// TIA Portal V15.1 export
// export: Created 2020-06-12T07:35:48.3037109Z, ExportSetting None, DisplayName Totally Integrated Automation Portal, DisplayVersion V15.1, DisplayName TIA Portal Openness, DisplayVersion V15.1, DisplayName STEP 7 Professional, DisplayVersion V15.1, DisplayName STEP 7 Safety, DisplayVersion V15.1, DisplayName WinCC Advanced, DisplayVersion V15.1
FUNCTION "PWR_ctrl" : Void   // FC751, FBD
TITLE = High current line
{ S7_Optimized_Access := 'TRUE' }
// stored: AutoNumber false, SetENOAutomatically False
   VAR_TEMP
      _dummy : Bool;
      _csf : Bool;   // Common system fault
      _trans_release : Bool;
      _mcb_lock : Bool;
      _mcb_start : Bool;
      _mcb_stop : Bool;
      _mcb_stop_cmd : Bool;
      _mcb_save_off : Bool;
      _slag_ok : Bool;
      _sealing_ok : Bool;
      _tp : Time;
      _toff : Bool;
      _spare : Bool;
      tRet : Int;
      tPmax : Real;
      tImax : Real;
      _mcb_released : Bool;
      tCbOn : Bool;
      tCosPhi : Real;
      tSwitchPulse : Bool;
      tCbExtOn : Bool;
      tCbExtOff : Bool;
      tCbIntOff : Bool;
      tCircuitInsulFault : Bool;
      tTrafoCoolFault : Bool;
      tCBisDisabled : Bool;
   END_VAR
BEGIN

REGION Network 1: Common System Fault
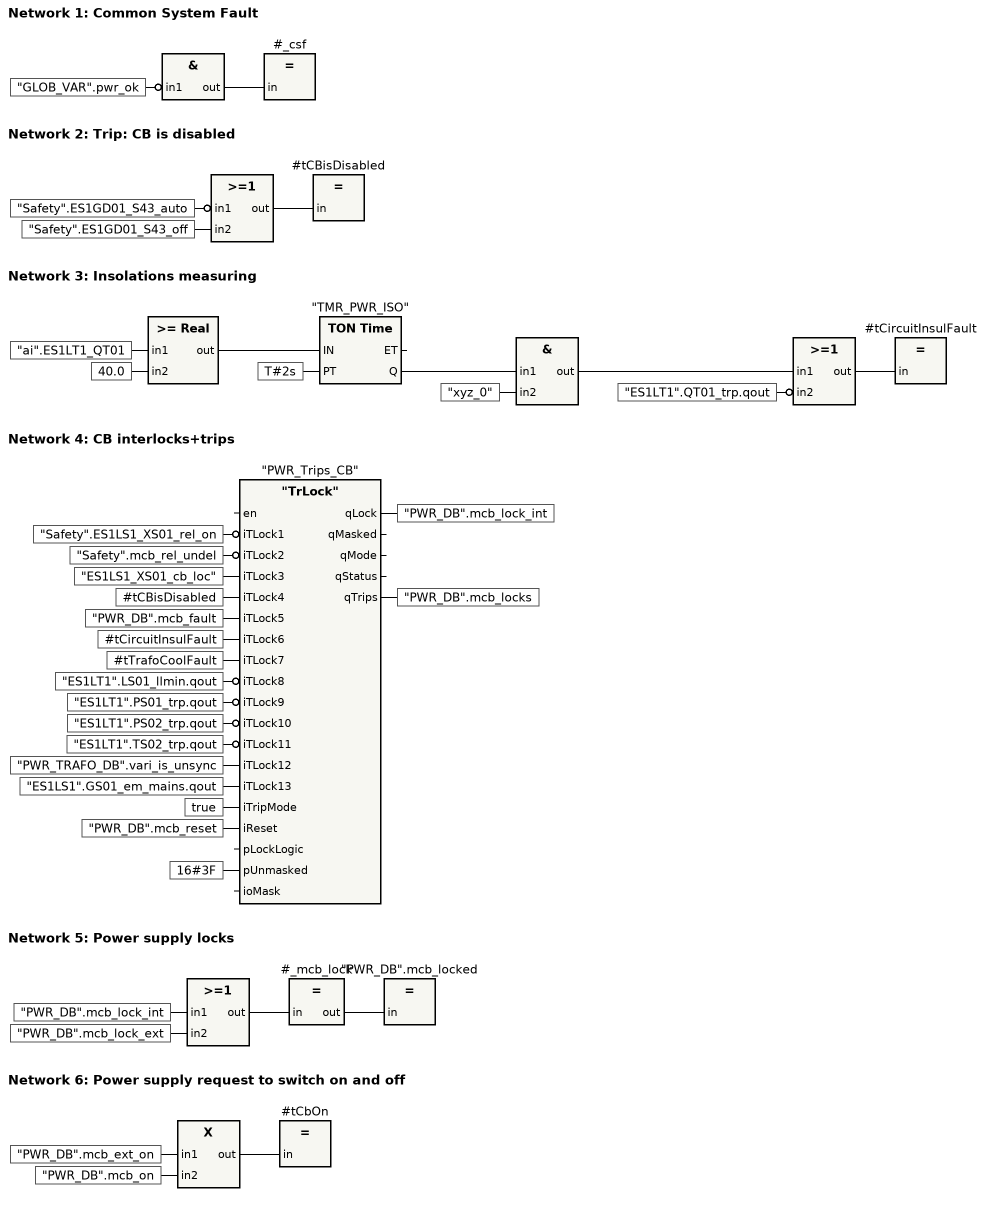
   #_csf := NOT "GLOB_VAR".pwr_ok;
END_REGION

REGION Network 2: Trip: CB is disabled
   #tCBisDisabled := NOT "Safety".ES1GD01_S43_auto OR "Safety".ES1GD01_S43_off;
END_REGION

REGION Network 3: Insolations measuring
   // "ES1LT1_QT01_ntrp"
   "TMR_PWR_ISO".TON(IN := "ai".ES1LT1_QT01 >= 40.0, PT := T#2s);
   #tCircuitInsulFault := ("TMR_PWR_ISO".Q AND "xyz_0") OR NOT "ES1LT1".QT01_trp.qout;
END_REGION

REGION Network 4: CB interlocks+trips
   // "PWR_DB".mcb_lock_int
   "PWR_Trips_CB"(iTLock1 := NOT "Safety".ES1LS1_XS01_rel_on,   // "TrLock"
                  iTLock2 := NOT "Safety".mcb_rel_undel,
                  iTLock3 := "ES1LS1_XS01_cb_loc",
                  iTLock4 := #tCBisDisabled,
                  iTLock5 := "PWR_DB".mcb_fault,
                  iTLock6 := #tCircuitInsulFault,
                  iTLock7 := #tTrafoCoolFault,
                  iTLock8 := NOT "ES1LT1".LS01_llmin.qout,
                  iTLock9 := NOT "ES1LT1".PS01_trp.qout,
                  iTLock10 := NOT "ES1LT1".PS02_trp.qout,
                  iTLock11 := NOT "ES1LT1".TS02_trp.qout,
                  iTLock12 := "PWR_TRAFO_DB".vari_is_unsync,
                  iTLock13 := "ES1LS1".GS01_em_mains.qout,
                  iTripMode := true,
                  iReset := "PWR_DB".mcb_reset,
                  pUnmasked := 16#3F,
                  qLock => "PWR_DB".mcb_lock_int,
                  qTrips => "PWR_DB".mcb_locks);
END_REGION

REGION Network 5: Power supply locks
   // !! NB: Ther are only physical locks which are not depend from the process conditions. But the process conditions are depend from the physical conditions.
   // PuM/2018-07-06: The signal "ES1LS1_XS01_cb_is_rdy" is using for interlock beacuse it means 'CB is charged'
   #_mcb_lock := "PWR_DB".mcb_lock_int OR "PWR_DB".mcb_lock_ext;
   "PWR_DB".mcb_locked := #_mcb_lock;
END_REGION

REGION Network 6: Power supply request to switch on and off
   #tCbOn := "PWR_DB".mcb_ext_on XOR "PWR_DB".mcb_on;
END_REGION

REGION Network 7: Main Circuit Breaker control
   // NOTE: MCB.iOn used as PULSE signal
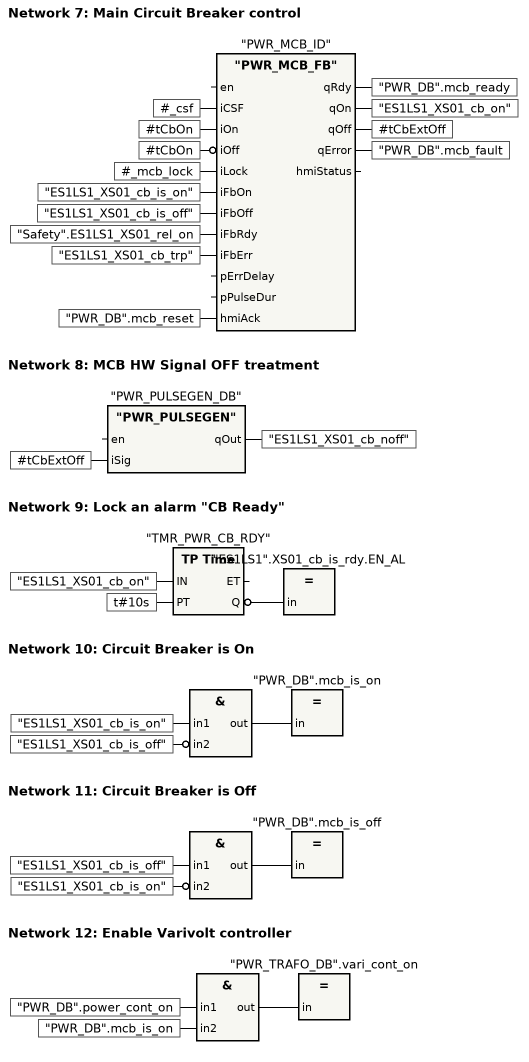
   "PWR_MCB_ID"(iCSF := #_csf,   // "PWR_MCB_FB"
                iOn := #tCbOn,
                iOff := NOT #tCbOn,
                iLock := #_mcb_lock,
                iFbOn := "ES1LS1_XS01_cb_is_on",
                iFbOff := "ES1LS1_XS01_cb_is_off",
                iFbRdy := "Safety".ES1LS1_XS01_rel_on,
                iFbErr := "ES1LS1_XS01_cb_trp",
                hmiAck := "PWR_DB".mcb_reset,
                qRdy => "PWR_DB".mcb_ready,
                qOn => "ES1LS1_XS01_cb_on",
                qOff => #tCbExtOff,
                qError => "PWR_DB".mcb_fault);
END_REGION

REGION Network 8: MCB HW Signal OFF treatment
   // By request of Mahesh I implement a one-shot pulse OFF signal.
   // But for me it looks not good, so I re-design the code and now a many-shot pluse OFF signal is using
   "PWR_PULSEGEN_DB"(iSig := #tCbExtOff, qOut => "ES1LS1_XS01_cb_noff");   // "PWR_PULSEGEN"
END_REGION

REGION Network 9: Lock an alarm "CB Ready"
   "TMR_PWR_CB_RDY".TP(IN := "ES1LS1_XS01_cb_on", PT := t#10s);
   "ES1LS1".XS01_cb_is_rdy.EN_AL := NOT "TMR_PWR_CB_RDY".Q;
END_REGION

REGION Network 10: Circuit Breaker is On
   "PWR_DB".mcb_is_on := "ES1LS1_XS01_cb_is_on" AND NOT "ES1LS1_XS01_cb_is_off";
END_REGION

REGION Network 11: Circuit Breaker is Off
   "PWR_DB".mcb_is_off := "ES1LS1_XS01_cb_is_off" AND NOT "ES1LS1_XS01_cb_is_on";
END_REGION

REGION Network 12: Enable Varivolt controller
   "PWR_TRAFO_DB".vari_cont_on := "PWR_DB".power_cont_on AND "PWR_DB".mcb_is_on;
END_REGION
END_FUNCTION
